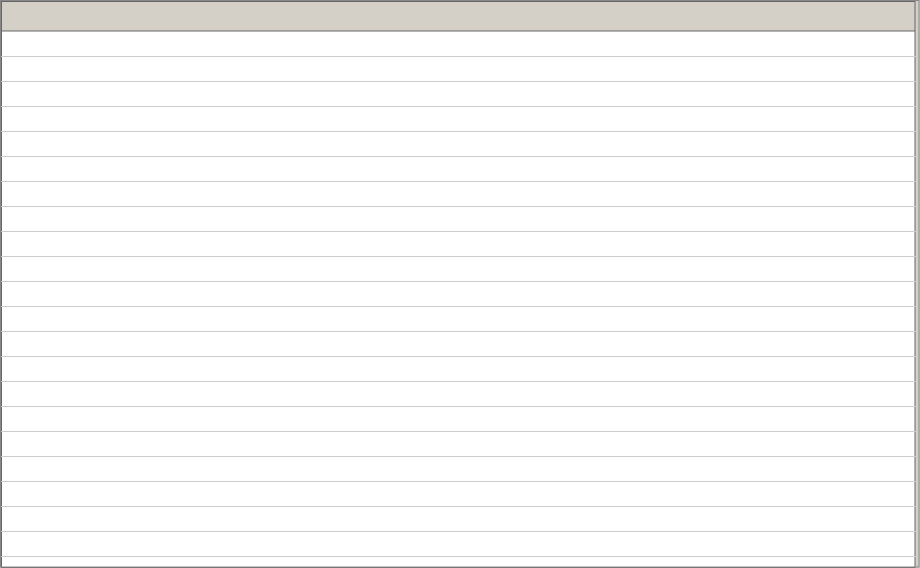
VISUALIZATION Alarm  // 920x568
    Table (1,1 914x567), data array: GVL_Retain.astAlarmHistory
        p3854506369: GVL_Retain.astAlarmHistory[INDEX].bActive
        p1892666644: GVL_Retain.astAlarmHistory[INDEX].iAlarmCode
        p338671338: GVL_Retain.astAlarmHistory[INDEX].sAlarmMessage
        p2170511999: GVL_Retain.astAlarmHistory[INDEX].tTimeStamp
        p3723444502: GVL_Retain.astAlarmHistory[INDEX].sLocation
        p1218418051: GVL_Retain.astAlarmHistory[INDEX].iPriority
        p4092479075: Time Stamp
        p1014161805: 99 - 0 + INT#1
        p1128707560: cMaxAlarmLogCount
END_VISUALIZATION

(* stored: Version 1.1.0.1
   Visu Alarm: Id {2617736b-a77d-4694-9809-35e53a3ed362} *)
